Staubli VAL3: HOME.pjx

--- HOME.pjx ---
Parameters version=s7.2.1 stackSize=5000 millimeterUnit=true
Data file=HOME.dtx
Library alias=io path=Disk://io/io.pjx

--- HOME.dtx ---
public num distance
public num moveType
public num nIndexGun
public num nTime
public num nStop
public num nTcpAction
public num nFrameIndex
public num nLaserPower
public num nGasPressure
public num nPWMPercent
public num nJointMode
public string comment
public string instruction
public string sProgram
public bool toStop
public frame fTrack = {fatherId=world[0]}
public jointRx jJoints
public mdesc nom_speed = {vel=10, tmax=9999, rmax=9999, leave=30, reach=30}
